Staubli VAL3: start.pgx

public program start()
begin
  if prog:libLoad("./Prog1")!=0
    logMsg("Error Loading RoboDK library")
    popUpMsg("Error Loading RoboDK library")
  endIf
  wait(taskStatus("loading")==-1)
  prog:fPartReal.trsf=fPartCad.trsf*fCadToReal.trsf
  prog:tCad.trsf=prog:tCad.trsf*{0,0,tooldata:nLength,0,0,0}
  call prog:start()


end
